{attribute 'GeneratedUsingTerminal: EL3692-0000-0017'}
{attribute addProperty BoxType "EL3692-0000-0017"}
{attribute addProperty Id "EtcSlaveTerminalBaseSAI_Inputs_Channel_1AT %I*SAI_Inputs_Channel_9DCD655714SAI_Range_Channel_1AT %I*SAI_Range_Channel_BDBF6DA92SAI_Inputs_Real_Channel_1AT %I*SAI_Inputs_Real_Channel_CCECF13D4SAI_Inputs_Channel_2AT %I*SAI_Inputs_Channel_9DCD655714SAI_Range_Channel_2AT %I*SAI_Range_Channel_BDBF6DA92SAI_Inputs_Real_Channel_2AT %I*SAI_Inputs_Real_Channel_CCECF13D4WcStateAT %I*WcState_9091E0EB2InfoDataAT %I*InfoData_32EB74EA10"}
{attribute addProperty CRC "3444495091"}
{attribute addProperty Size "52"}
TYPE EL3692_CD4ED2F3 EXTENDS EtcSlaveTerminalBase :
STRUCT
	{attribute addProperty Name "SAI_Inputs_Channel_1"}
	SAI_Inputs_Channel_1 : SAI_Inputs_Channel_9DCD6557;
	{attribute addProperty Name "SAI_Range_Channel_1"}
	SAI_Range_Channel_1 : SAI_Range_Channel_BDBF6DA9;
	{attribute addProperty Name "SAI_Inputs_Real_Channel_1"}
	SAI_Inputs_Real_Channel_1 : SAI_Inputs_Real_Channel_CCECF13D;
	{attribute addProperty Name "SAI_Inputs_Channel_2"}
	SAI_Inputs_Channel_2 : SAI_Inputs_Channel_9DCD6557;
	{attribute addProperty Name "SAI_Range_Channel_2"}
	SAI_Range_Channel_2 : SAI_Range_Channel_BDBF6DA9;
	{attribute addProperty Name "SAI_Inputs_Real_Channel_2"}
	SAI_Inputs_Real_Channel_2 : SAI_Inputs_Real_Channel_CCECF13D;
	{attribute addProperty Name "WcState"}
	WcState : WcState_9091E0EB;
	{attribute addProperty Name "InfoData"}
	InfoData : InfoData_32EB74EA;
END_STRUCT
END_TYPE

(* stored: Version 1.2.0.0, ProductVersion 3.1.4024.9
   DUT EL3692_CD4ED2F3: Id {9cff1467-ada0-43bb-90cb-a56df8b15879} *)
